FUNCTION_BLOCK T_NotificationHandler IMPLEMENTS I_NotificationHandler
VAR
    Args_LocalCopy      : T_Stream(StreamLength := 4); // Local copy of notification arguments
    Args_PublicCopy     : T_Stream(StreamLength := 4); // Public copy of notification arguments
    CriticalSection     : FB_IecCriticalSection;
    NotificationCounter : T_Counter;
    QueueingEnabled     : BOOL; // if required, set via variable initialisation in instance declaration
END_VAR
VAR CONSTANT
    MAX_UNHANDLED_NOTIFICATIONS : DINT := 1000;
END_VAR

PROPERTY Args : I_StreamReader
GET
Args := Args_PublicCopy;
END_GET
END_PROPERTY

METHOD IsRaised : BOOL
VAR
    ByteCount : UDINT;
END_VAR
IF CriticalSection.hrInit = S_OK THEN
    IF CriticalSection.Enter() THEN           // will block while receiving a notification
        IF NotificationCounter.Value > 0 THEN // at least one unhandled notification to be handled...
            IsRaised := TRUE;

            // get the length of the notification args (this is stored before the args themselves)
            ByteCount := Args_LocalCopy.Read_UDINT();

            // Copy the args for this notification to the public copy of the args, which can be accessed externally...
            Args_PublicCopy.Clear();
            Args_PublicCopy.AppendBytesFromStream(Args_LocalCopy,
                                                  ByteCount);

            NotificationCounter.Dec(); // to keep track of how many notifications remain to be handled

            IF NotificationQueueingEnabled AND NotificationCounter.Value > 0 THEN // more args to be handled (notification raised multiple times since last handled)...
                // advance the read pointer to the args belonging to the next notification (if any)                                      
                Args_LocalCopy.SetReadPosition(Args_LocalCopy.ReadPosition + ByteCount);
            ELSE // clear any unhandled notifications that remain..
				NotificationCounter.Reset();
                Args_LocalCopy.Clear();
            END_IF
        END_IF

        CriticalSection.Leave();
    END_IF
ELSE
    F_LogError(Source := 'T_NotificationHandler', Message := 'FB_IEC_CriticalSection not initialised!');
END_IF
END_METHOD

PROPERTY NotificationCount : DINT
GET
NotificationCount := NotificationCounter.Value;
END_GET
END_PROPERTY

PROPERTY NotificationQueueingEnabled : BOOL// Allows notifications to be raised multiple times before being handled sequentially. Make sure all notifications are handled!
GET
NotificationQueueingEnabled := QueueingEnabled;
END_GET
SET
QueueingEnabled := NotificationQueueingEnabled;
END_SET
END_PROPERTY

METHOD RaiseNotification
VAR_INPUT
    NotificationArgs : I_StreamReader;
END_VAR
IF NotificationCounter.Value > MAX_UNHANDLED_NOTIFICATIONS THEN
    // Not much point raising another if they are not being handled...
    RETURN;
END_IF

IF CriticalSection.Enter() THEN
    IF NotificationArgs.WritePosition > 0 THEN // has event arguments..

        // Notification args are stored in a local copy using a stream
        // If the notification is raised again before being handled, the newer notification args are just added to the stream
        // The size of the args is stored in the stream before the args themselves so they
        // can be retrieved seperately when the notifications are handled    

        Args_LocalCopy.Add_UDINT(NotificationArgs.WritePosition); // length of args is stored first
        Args_LocalCopy.AppendBytesFromStream(StreamToAppend        := NotificationArgs,
                                             NumberOfBytesToAppend := NotificationArgs.WritePosition); // followed by args themselves
    END_IF

    NotificationCounter.Inc(); // keep track of how many times the notification has been raised, so we can handle each notification seperately
    CriticalSection.Leave();
END_IF
END_METHOD

END_FUNCTION_BLOCK

(* stored: Version 1.1.0.1, ProductVersion 3.1.4024.12
   POU T_NotificationHandler: Id {607f5e14-d01e-4493-979d-0fc6e8f214bb}, SpecialFunc None
   Folder Methods: Id {50523a27-f4f0-421d-b359-9106ca91093f}
   Folder Properties: Id {bcb797de-c3f3-40e6-aa20-89bbc5f8f950}
   Property Args: Id {677afeaa-0697-40f0-93b0-2ba305384c9c}
   Get Get: Id {3597fd34-9332-43bd-a3f4-c1cacf585b03}
   Method IsRaised: Id {e8102458-838e-441a-8b86-1d3da0b59390}
   Property NotificationCount: Id {75289af6-a460-4022-ac06-0483ce39413a}
   Get Get: Id {80a90d77-9dc4-4e7c-a8ec-f0f39e5d20cc}
   Property NotificationQueueingEnabled: Id {a5314985-f357-4fe9-a599-bc37bf9428ff}
   Get Get: Id {1b6498ce-791f-4589-943b-9a1edc56d6b6}
   Set Set: Id {3bfda8f6-68ff-4cb0-9193-8ace86f621f9}
   Method RaiseNotification: Id {8767452b-6194-4156-b4a1-080cf2d33e36} *)
